FUNCTION_BLOCK GF_Pumpen EXTENDS FB_Basis
VAR_INPUT
	// Instanzieren von Sensoren mit Interfaces
	
	// Instanzieren von Aktoren mit Interfaces
	Ventil_IN			:I_Magnetventil;
	Ventil_OUT			:I_Magnetventil;
	
	Pumpe				:I_Motor2R;
	
END_VAR
VAR_OUTPUT
	
END_VAR
VAR
	
END_VAR

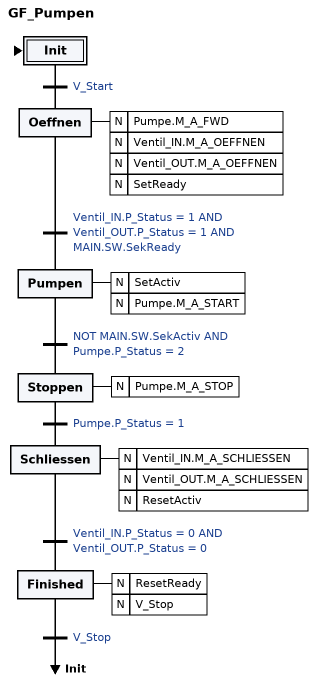
INITIAL_STEP Init:
END_STEP
TRANSITION FROM Init TO Oeffnen
    := V_Start;
END_TRANSITION
STEP Oeffnen:
    Pumpe.M_A_FWD(N);
    Ventil_IN.M_A_OEFFNEN(N);
    Ventil_OUT.M_A_OEFFNEN(N);
    SetReady(N);
END_STEP
TRANSITION FROM Oeffnen TO Pumpen
    := Ventil_IN.P_Status = 1 AND Ventil_OUT.P_Status = 1 AND MAIN.SW.SekReady;
END_TRANSITION
STEP Pumpen:
    SetActiv(N);
    Pumpe.M_A_START(N);
END_STEP
TRANSITION FROM Pumpen TO Stoppen
    := NOT MAIN.SW.SekActiv AND Pumpe.P_Status = 2;
END_TRANSITION
STEP Stoppen:
    Pumpe.M_A_STOP(N);
END_STEP
TRANSITION FROM Stoppen TO Schliessen
    := Pumpe.P_Status = 1;
END_TRANSITION
STEP Schliessen:
    Ventil_IN.M_A_SCHLIESSEN(N);
    Ventil_OUT.M_A_SCHLIESSEN(N);
    ResetActiv(N);
END_STEP
TRANSITION FROM Schliessen TO Finished
    := Ventil_IN.P_Status = 0 AND Ventil_OUT.P_Status = 0;
END_TRANSITION
STEP Finished:
    ResetReady(N);
    V_Stop(N);
END_STEP
TRANSITION FROM Finished TO Init
    := V_Stop;
END_TRANSITION

ACTION ResetActiv:
MAIN.SW.PrimActiv := FALSE;
END_ACTION

ACTION ResetReady:
MAIN.SW.PrimReady := FALSE;
END_ACTION

ACTION SetActiv:
MAIN.SW.PrimActiv := TRUE;
END_ACTION

ACTION SetReady:
MAIN.SW.PrimReady := TRUE;
END_ACTION

END_FUNCTION_BLOCK

(* stored: Version 1.1.0.1, ProductVersion 3.1.4024.12
   POU GF_Pumpen: Id {298b1c00-eb4e-4c76-a60a-3efaa29ca07f}, SpecialFunc None
   Folder 01_Aktionen: Id {6dd232fd-6ffa-44e2-a3a0-37b9dcd0166e}
   Action ResetActiv: Id {c3fbeb30-5f5e-4a38-b89a-e5470edfd818}
   Action ResetReady: Id {19e5b31a-746d-4074-9b95-d00e50531829}
   Action SetActiv: Id {78df1253-aaa8-4459-8da8-af86452c84a0}
   Action SetReady: Id {aebbd464-42ad-42e3-bb8f-c2e8c80694d7} *)
